TEXTLIST TL_SelectedParameterSet
  0 = 'Fast'
  1 = 'Slow'
  2 = 'Asymptotic'
   = ''
END_TEXTLIST

(* stored: Version 1.1.0.1, ProductVersion 3.1.4024.12
   TextList TL_SelectedParameterSet: Id {9746303c-ff39-44e9-a49a-ce12d20a8341} *)
